FUNCTION_BLOCK TrackFactory EXTENDS Factory
VAR
	ptrTrack : POINTER TO Track;
	itfTrack : ITF_Track;
END_VAR

METHOD Create : ITF_Cyclic
VAR_INPUT
END_VAR
ptrTrack := __NEW(Track);
Create := ptrTrack^;
IF __QUERYINTERFACE(Create,itfTrack) THEN
	itfTrack.Length := 2500.0;
END_IF
END_METHOD

END_FUNCTION_BLOCK

(* stored: Version 1.1.0.1, ProductVersion 3.1.4024.12
   POU TrackFactory: Id {ec46e399-6229-4d9f-9958-4db80a70545f}, SpecialFunc None
   Method Create: Id {821dd5c5-4056-4ccc-a667-62f25eca92dd} *)
